// TIA Portal V18 export
FUNCTION_BLOCK "FC51_Modbus_Com"   // FB101, LAD
{ S7_Optimized_Access := 'FALSE' }
// stored: SetENOAutomatically false
   VAR_INPUT
      I_Modbus_Slave_Addr : Byte;
      I_Start : Bool;
      I_Reset : Bool;
      I_Ramp_Switch : Bool;   // 0: Ramp 1, 1: Ramp2
      I_Relay_1 : Bool;
      I_Frequency : Word;   // 0-100（%）
   END_VAR
   VAR
      FB_Always_True : Bool;
      Modbus_DATA : Array[0..1] of Word;
      Ctrl_Bits : Array[1..32] of Bool;
      Gateway_IP { ExternalAccessible := 'False'; ExternalVisible := 'False'; ExternalWritable := 'False'} : TCON_IP_v4;
      MB_CLIENT_Instance : MB_CLIENT;
   END_VAR
   // Gateway_IP.InterfaceId := 64;
   // Gateway_IP.ID := 2;
   // Gateway_IP.ActiveEstablished := TRUE;
   // Gateway_IP.RemoteAddress.ADDR[1] := 192;
   // Gateway_IP.RemoteAddress.ADDR[2] := 168;
   // Gateway_IP.RemoteAddress.ADDR[3] := 6;
   // Gateway_IP.RemoteAddress.ADDR[4] := 11;
   // Gateway_IP.RemotePort := 502;
   // Gateway_IP.LocalPort := 0;
BEGIN

REGION Network 1: FBAT
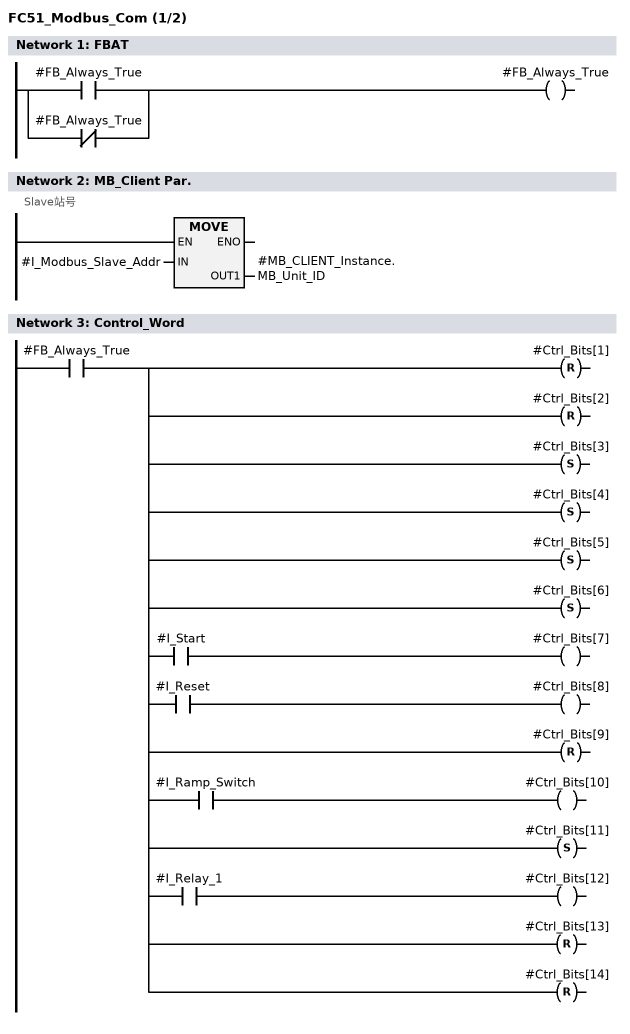
   RUNG wire#powerrail
      Contact( #FB_Always_True )
      wire#w1
      Coil( #FB_Always_True )
   END_RUNG
   RUNG wire#powerrail
      I_Contact( #FB_Always_True )
   END_RUNG wire#w1
   // the same network as SCL:
   #FB_Always_True := #FB_Always_True OR NOT #FB_Always_True;
END_REGION

REGION Network 2: MB_Client Par.
   // Slave站号
   RUNG wire#powerrail
      Move(in := #I_Modbus_Slave_Addr, out1 => #MB_CLIENT_Instance.MB_Unit_ID)
   END_RUNG
   // the same network as SCL:
   #MB_CLIENT_Instance.MB_Unit_ID := #I_Modbus_Slave_Addr;
END_REGION

REGION Network 3: Control_Word
   RUNG wire#powerrail
      Contact( #FB_Always_True )
      wire#w1
      R_Coil( #Ctrl_Bits[1] )
   END_RUNG
   RUNG wire#w1
      R_Coil( #Ctrl_Bits[2] )
   END_RUNG
   RUNG wire#w1
      S_Coil( #Ctrl_Bits[3] )
   END_RUNG
   RUNG wire#w1
      S_Coil( #Ctrl_Bits[4] )
   END_RUNG
   RUNG wire#w1
      S_Coil( #Ctrl_Bits[5] )
   END_RUNG
   RUNG wire#w1
      S_Coil( #Ctrl_Bits[6] )
   END_RUNG
   RUNG wire#w1
      Contact( #I_Start )
      Coil( #Ctrl_Bits[7] )
   END_RUNG
   RUNG wire#w1
      Contact( #I_Reset )
      Coil( #Ctrl_Bits[8] )
   END_RUNG
   RUNG wire#w1
      R_Coil( #Ctrl_Bits[9] )
   END_RUNG
   RUNG wire#w1
      Contact( #I_Ramp_Switch )
      Coil( #Ctrl_Bits[10] )
   END_RUNG
   RUNG wire#w1
      S_Coil( #Ctrl_Bits[11] )
   END_RUNG
   RUNG wire#w1
      Contact( #I_Relay_1 )
      Coil( #Ctrl_Bits[12] )
   END_RUNG
   RUNG wire#w1
      R_Coil( #Ctrl_Bits[13] )
   END_RUNG
   RUNG wire#w1
      R_Coil( #Ctrl_Bits[14] )
   END_RUNG
   // the same network as SCL:
   IF #FB_Always_True THEN
       #Ctrl_Bits[1] := FALSE;
       #Ctrl_Bits[2] := FALSE;
       #Ctrl_Bits[3] := TRUE;
       #Ctrl_Bits[4] := TRUE;
       #Ctrl_Bits[5] := TRUE;
       #Ctrl_Bits[6] := TRUE;
   END_IF;
   #Ctrl_Bits[7] := #FB_Always_True AND #I_Start;
   #Ctrl_Bits[8] := #FB_Always_True AND #I_Reset;
   IF #FB_Always_True THEN #Ctrl_Bits[9] := FALSE; END_IF;
   #Ctrl_Bits[10] := #FB_Always_True AND #I_Ramp_Switch;
   IF #FB_Always_True THEN #Ctrl_Bits[11] := TRUE; END_IF;
   #Ctrl_Bits[12] := #FB_Always_True AND #I_Relay_1;
   IF #FB_Always_True THEN
       #Ctrl_Bits[13] := FALSE;
       #Ctrl_Bits[14] := FALSE;
   END_IF;
END_REGION

REGION Network 4 (SCL): Frequency Input
   #Modbus_DATA[1] := #I_Frequency;
END_REGION

REGION Network 5: Control_Word
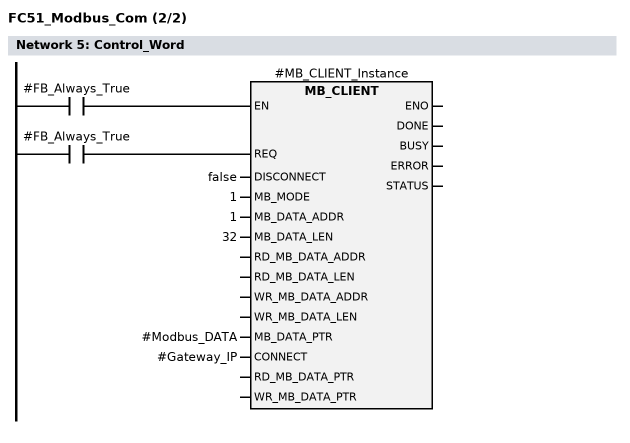
   RUNG wire#powerrail
      Contact( #FB_Always_True )
      #MB_CLIENT_Instance.MB_CLIENT(REQ := wire#w1, DISCONNECT := false, MB_MODE := 1, MB_DATA_ADDR := 1, MB_DATA_LEN := 32, RD_MB_DATA_ADDR :=, RD_MB_DATA_LEN :=, WR_MB_DATA_ADDR :=, WR_MB_DATA_LEN :=, MB_DATA_PTR := #Modbus_DATA, CONNECT := #Gateway_IP, RD_MB_DATA_PTR :=, WR_MB_DATA_PTR :=, DONE =>, BUSY =>, ERROR =>, STATUS =>)
   END_RUNG
   RUNG wire#powerrail
      Contact( #FB_Always_True )
   END_RUNG wire#w1
   // the same network as SCL:
   IF #FB_Always_True THEN
       #MB_CLIENT_Instance(REQ := #FB_Always_True,   // MB_CLIENT
                           DISCONNECT := false,
                           MB_MODE := 1,
                           MB_DATA_ADDR := 1,
                           MB_DATA_LEN := 32,
                           MB_DATA_PTR := #Modbus_DATA,
                           CONNECT := #Gateway_IP);
   END_IF;
END_REGION
END_FUNCTION_BLOCK
